Yaskawa INFORM job: SYS_UNLOCK_GATE.JBI

/JOB
//NAME SYS_UNLOCK_GATE
//POS
///NPOS 0,0,0,0,0,0
//INST
///DATE 2022/05/18 13:57
///ATTR SC,RW
///GROUP1 RB1
NOP
DOUT OT#(19) ON
END
